PROGRAM AST40_Controller
VAR
END_VAR

END_PROGRAM

(* stored: Version 1.1.0.1, ProductVersion 3.1.4022.18
   POU AST40_Controller: Id {1db48b83-1c1e-4170-aa6c-e6f8192c6e0f}, SpecialFunc None *)
